FUNCTION_BLOCK INTEGRAL (* determines approximately the integral over time. *)
  (* Standard: 61499-1; Description: Copyright (c) 2024 HR Agrartechnik GmbH This program and the accompanying materials are made available under the terms of the Eclipse Public License 2.0 which is available at https://www.eclipse.org/legal/epl-2.0/ SPDX-License-Identifier: EPL-2.0 This Block was inspired by https://content.helpme-codesys.com/en/libs/Util/Current/Mathematical-Functions/INTEGRAL.html *)
  (* Version 1.0, 2024-10-18, franz *)
  PACKAGE utils::math;
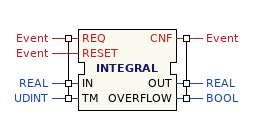
  EVENT_INPUT
    REQ WITH IN, TM; (* Normal Execution Request *)
    RESET; (* TRUE: OUT is set to zero and OVERFLOW to FALSE *)
  END_EVENT
  EVENT_OUTPUT
    CNF WITH OUT, OVERFLOW; (* Execution Confirmation *)
  END_EVENT
  VAR_INPUT
    IN : REAL; (* Input value *)
    TM : UDINT; (* Time since last call in msec *)
  END_VAR
  VAR_OUTPUT
    OUT : REAL; (* Value of the integral. This is done by summing all part integrals IN * TM *)
    OVERFLOW : BOOL; (* TRUE: The value of OUT is out of range of REAL variables. he function is blocked till it is new initialised by input RESET. *)
  END_VAR
  ALGORITHM REQ IN ST:
IF NOT OVERFLOW THEN
	IF (1.0E38 - IN * UDINT_TO_REAL(TM) < OUT OR -1.0E38 - IN * UDINT_TO_REAL(TM) > OUT) THEN
		OVERFLOW := TRUE;
	ELSE
		OUT := OUT + IN * UDINT_TO_REAL(TM) / 1000.0;

	END_IF;
END_IF;
  END_ALGORITHM
  ALGORITHM RESET IN ST:
OUT := 0.0;
OVERFLOW := FALSE;
  END_ALGORITHM
END_FUNCTION_BLOCK
